FUNCTION_BLOCK ASSEMBLE_AL_FROM_AD (* this Function combines the 2 AD (DWORD) adapters to a AL (LWORD) *)
  (* Standard: 61499-2; Description: Copyright (c) 2026 Meisterschulen am Ostbahnhof SPDX-License-Identifier: EPL-2.0 *)
  (* Version 1.0, 2026-05-16, Franz Höpfinger, Meisterschulen am Ostbahnhof, initial API and implementation and/or initial documentation *)
  PACKAGE adapter::assembling;
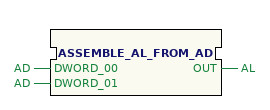
  SOCKETS
    DWORD_00 : adapter::types::unidirectional::AD; (* DWord 0 *)
    DWORD_01 : adapter::types::unidirectional::AD; (* DWord 1 *)
  END_SOCKETS
  PLUGS
    OUT : adapter::types::unidirectional::AL; (* LWORD Output *)
  END_PLUGS
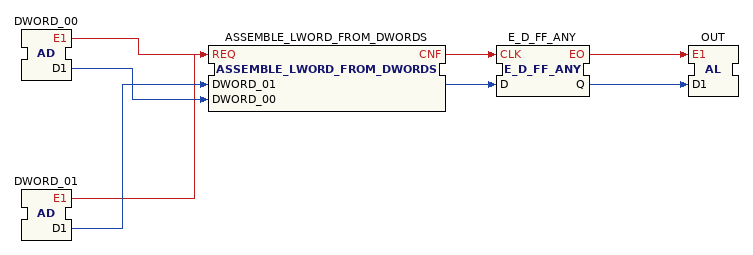
  FBS
    ASSEMBLE_LWORD_FROM_DWORDS : eclipse4diac::utils::assembling::ASSEMBLE_LWORD_FROM_DWORDS;
    E_D_FF_ANY : iec61499::events::E_D_FF_ANY;
  END_FBS
  EVENT_CONNECTIONS
    DWORD_00.E1 TO ASSEMBLE_LWORD_FROM_DWORDS.REQ;
    DWORD_01.E1 TO ASSEMBLE_LWORD_FROM_DWORDS.REQ;
    ASSEMBLE_LWORD_FROM_DWORDS.CNF TO E_D_FF_ANY.CLK;
    E_D_FF_ANY.EO TO OUT.E1;
  END_CONNECTIONS
  DATA_CONNECTIONS
    ASSEMBLE_LWORD_FROM_DWORDS. TO E_D_FF_ANY.D;
    E_D_FF_ANY.Q TO OUT.D1;
    DWORD_01.D1 TO ASSEMBLE_LWORD_FROM_DWORDS.DWORD_01;
    DWORD_00.D1 TO ASSEMBLE_LWORD_FROM_DWORDS.DWORD_00;
  END_CONNECTIONS
END_FUNCTION_BLOCK
